ABB RobotStudio station: Moving_Conveyor.rsstn

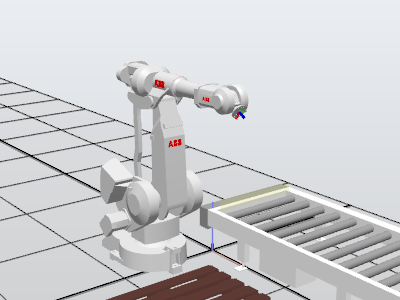
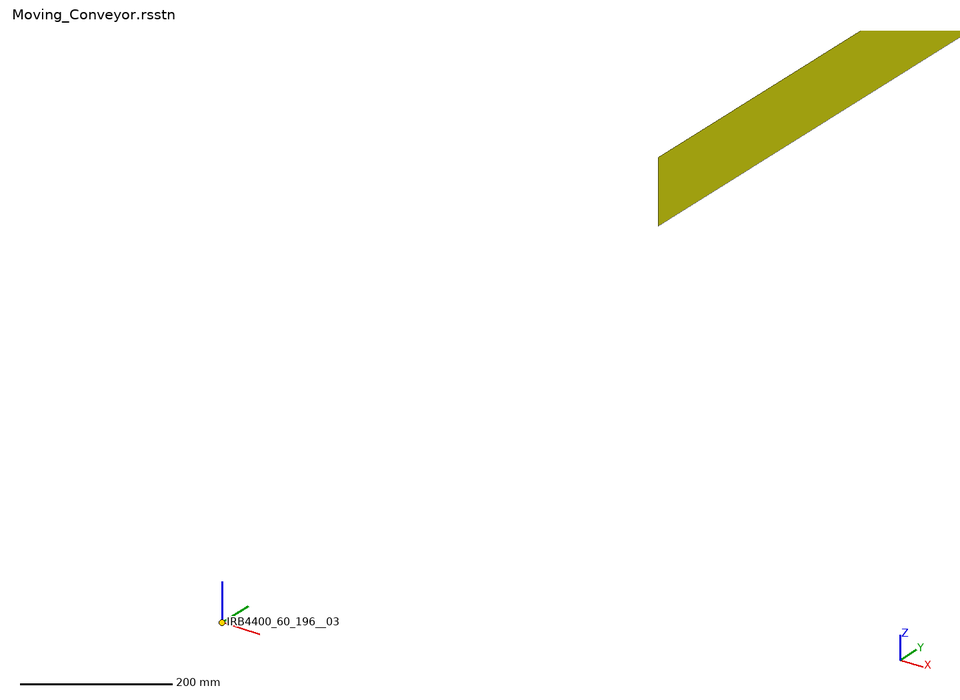
[picture v1: parts stored in the station drawn from their meshes, with robot base, taught points and paths (robot models come from the ABB library and are not in the file)]
Station Moving_Conveyor (saved by RobotStudio 24.3.10958.1)
Controller Controller26, task T_ROB1: task frame (RAPID world) sits at (-191.06, -562.78, 0) mm in the station
Controller Controller26
  mechanical unit ROB_1: IRB4400_60_196__03, 6 joints, base frame (0, 0, 0) mm
Layout (positions relative to the parent item):
  - SC_FeedingConveyor [smart component]
      signals: DI Turn_Conveyor_On, DO Conveyor_Complete
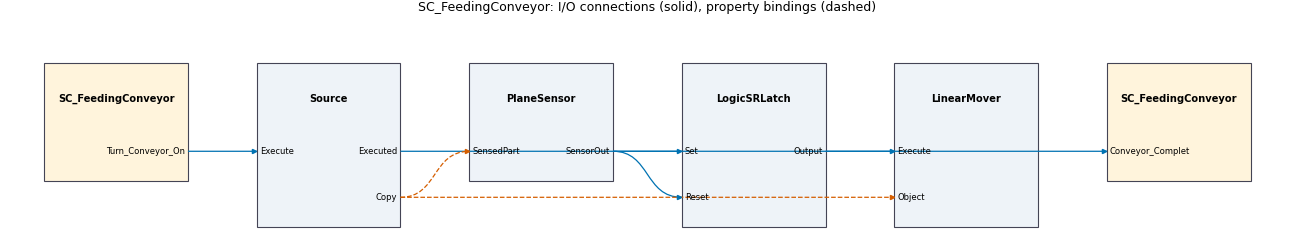
      connections:
        SC_FeedingConveyor.Turn_Conveyor_On -> Source.Execute
        Source.Executed -> LogicSRLatch.Set
        LogicSRLatch.Output -> LinearMover.Execute
        PlaneSensor.SensorOut -> LogicSRLatch.Reset
        PlaneSensor.SensorOut -> SC_FeedingConveyor.Conveyor_Complete
        Source.Copy => LinearMover.Object
        Source.Copy => PlaneSensor.SensedPart
    - LinearMover [smart component, from Components\LinearMover.rslib]
        properties: Object=(none); Direction=[-1 0 0]; Speed=0.5; Reference=Global; ReferenceObject=(none)
    - Source [smart component, from Components\Source.rslib]
        properties: Source=Part_1; Copy=(none); Parent=(none); Position=[3.775839 0.349686 0.420766]; Orientation=[0 0 0]; Transient=false; PhysicsBehavior=0
    - LogicSRLatch [smart component, from Components\LogicSRLatch.rslib]
    - PlaneSensor [smart component, from Components\PlaneSensor.rslib] at (108.31, 4.96, 897.38) mm
        properties: Origin=[0 0 -0.462381201751226]; Axis1=[0 0.9 0]; Axis2=[0 0 0.1]; Tag=(none); SensedPart=(none)
      - _sensorPart_ [part], size 0 x 900 x 100 mm
    - 950_4000_h2 [part, from %ABB.RobotStudio.Models.Conveyors%\Conveyor 950 4000 h2.rslib]
    - Part_1 [part] at (3775.84, 349.69, 420.77) mm, size 200 x 200 x 200 mm
  - IRB4400_60_196__03 [mechanism, from %ABB.RobotStudio.Models.IRB4400%\IRB4400_60_196_G_03.rslib] at (-191.06, -562.78, 0) mm; joint values [0, 0, 0, 0, 0.5236, 0] (rad or m)
  - Euro Pallet [graphiccomponentgroup, from Equipment\Euro Pallet.rslib] at (476, -410, 0) mm, rotated rx 0 ry 0 rz -90 deg
    - Body 1 [part, from Equipment\Euro Pallet.rslib]
